FUNCTION_BLOCK A2X2_2AX2_TO_2X (* Composite FB for convert 2 AX2 to A2X2 *)
  (* Standard: 61499-2; Description: Copyright (c) 2026 HR Agrartechnik GmbH This program and the accompanying materials are made available under the terms of the Eclipse Public License 2.0 which is available at https://www.eclipse.org/legal/epl-2.0/ SPDX-License-Identifier: EPL-2.0 *)
  (* Version 1.0, 2026-08-31, Franz Höpfinger, HR Agrartechnik GmbH *)
  PACKAGE adapter::conversion::bidirectional;
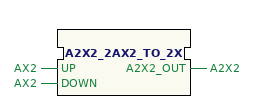
  SOCKETS
    UP : adapter::types::bidirectional::AX2; (* TRUE = forward, up, right, clockwise *)
    DOWN : adapter::types::bidirectional::AX2; (* TRUE = backward, down, left, counter-clockwise *)
  END_SOCKETS
  PLUGS
    A2X2_OUT : adapter::types::bidirectional::A2X2; (* Adapter Output *)
  END_PLUGS
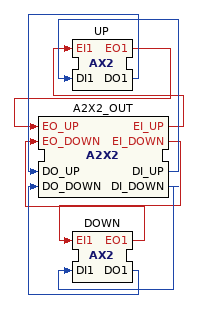
  EVENT_CONNECTIONS
    A2X2_OUT.EI_UP TO UP.EI1;
    UP.EO1 TO A2X2_OUT.EO_UP;
    A2X2_OUT.EI_DOWN TO DOWN.EI1;
    DOWN.EO1 TO A2X2_OUT.EO_DOWN;
  END_CONNECTIONS
  DATA_CONNECTIONS
    A2X2_OUT.DI_UP TO UP.DI1;
    UP.DO1 TO A2X2_OUT.DO_UP;
    A2X2_OUT.DI_DOWN TO DOWN.DI1;
    DOWN.DO1 TO A2X2_OUT.DO_DOWN;
  END_CONNECTIONS
END_FUNCTION_BLOCK
